PROGRAM MAIN
VAR
END_VAR

END_PROGRAM

(* stored: Version 1.1.0.1
   POU MAIN: Id {956d7ef0-483a-4ef2-94d3-858d4365b4a7} *)
